SUBAPPLICATION Q_ChildPosition_AR_Vertikal (* Command change child position (Y via AR adapter, X fixed to 0) *)
  (* Standard: 61499-2; Description: Copyright (c) 2026 Meisterschulen am Ostbahnhof This program and the accompanying materials are made available under the terms of the Eclipse Public License 2.0 which is available at https://www.eclipse.org/legal/epl-2.0/ SPDX-License-Identifier: EPL-2.0 *)
  (* Version 1.0, 2026-09-27, Franz Höpfinger, Meisterschulen am Ostbahnhof, initial API and implementation: AR adapter input to Y position, X fixed to 0 (AR_TO_AI + initval_AI + Q_ChildPosition_AI) *)
  PACKAGE MyLib::sys;
  IMPORT isobus::UT::Q::Q_ChildPosition_AI;
  IMPORT isobus::UT::Q::const::IDs::ID_NULL;
  IMPORT adapter::conversion::unidirectional::AR_TO_AI;
  IMPORT adapter::types::unidirectional::AI::initval::initval_AI;
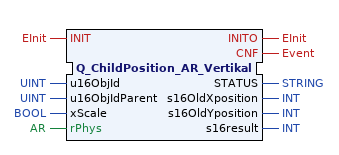
  EVENT_INPUT
    INIT : EInit; (* Service Initialization *)
  END_EVENT
  EVENT_OUTPUT
    INITO : EInit; (* Initialization Confirm *)
    CNF; (* Confirmation of Requested Service *)
  END_EVENT
  VAR_INPUT
    u16ObjId : UINT := ID_NULL; (* Object ID *)
    u16ObjIdParent : UINT := ID_NULL; (* Parent object ID *)
    xScale : BOOL := FALSE; (* FALSE (default) = bypass, send s16Xposition/s16Yposition through unchanged. TRUE = scale them by the DM/SKM factor for u16ObjIdParent. *)
  END_VAR
  VAR_OUTPUT
    STATUS : STRING; (* Service Status - passthrough from the internal Q_ChildPosition *)
    s16OldXposition : INT; (* Old X position - passthrough from the internal Q_ChildPosition *)
    s16OldYposition : INT; (* Old Y position - passthrough from the internal Q_ChildPosition *)
    s16result : INT; (* retval - passthrough from the internal Q_ChildPosition, see Q_ChildPosition *)
  END_VAR
  SOCKETS
    rPhys : adapter::types::unidirectional::AR; (* Physical REAL value input (converted to INT and mapped to Y position) *)
  END_SOCKETS
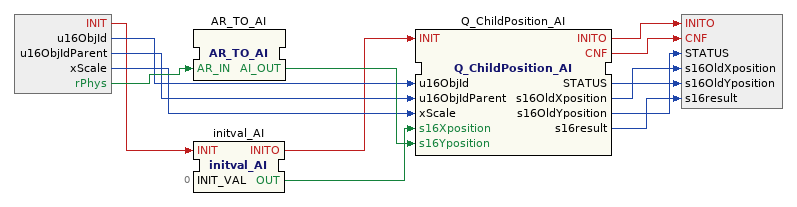
  FBS
    AR_TO_AI : adapter::conversion::unidirectional::AR_TO_AI;
    initval_AI : adapter::types::unidirectional::AI::initval::initval_AI(INIT_VAL := 0);
    Q_ChildPosition_AI : isobus::UT::Q::Q_ChildPosition_AI;
  END_FBS
  EVENT_CONNECTIONS
    INIT TO initval_AI.INIT;
    initval_AI.INITO TO Q_ChildPosition_AI.INIT;
    Q_ChildPosition_AI.INITO TO INITO;
    Q_ChildPosition_AI.CNF TO CNF;
  END_CONNECTIONS
  DATA_CONNECTIONS
    u16ObjId TO Q_ChildPosition_AI.u16ObjId;
    u16ObjIdParent TO Q_ChildPosition_AI.u16ObjIdParent;
    xScale TO Q_ChildPosition_AI.xScale;
    Q_ChildPosition_AI.STATUS TO STATUS;
    Q_ChildPosition_AI.s16OldXposition TO s16OldXposition;
    Q_ChildPosition_AI.s16OldYposition TO s16OldYposition;
    Q_ChildPosition_AI.s16result TO s16result;
  END_CONNECTIONS
  ADAPTER_CONNECTIONS
    rPhys TO AR_TO_AI.AR_IN;
    initval_AI.OUT TO Q_ChildPosition_AI.s16Xposition;
    AR_TO_AI.AI_OUT TO Q_ChildPosition_AI.s16Yposition;
  END_CONNECTIONS
END_SUBAPPLICATION
